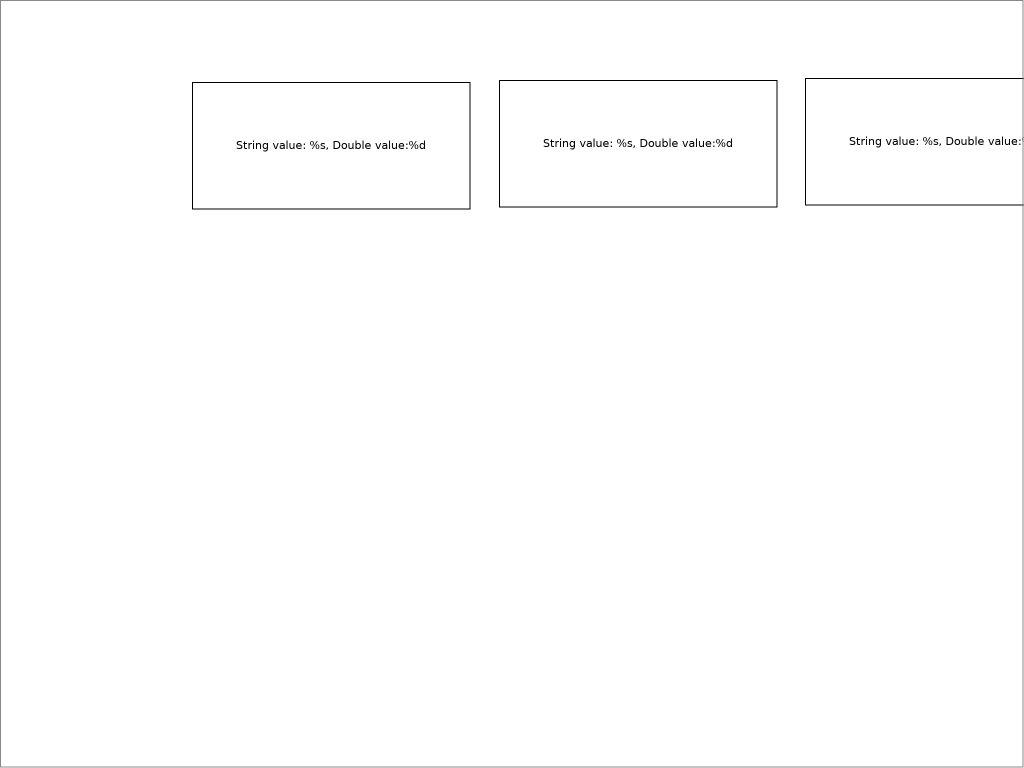
VISUALIZATION Visualization  // 1024x768
    Rectangle (192,82 278x127), "String value: %s, Double value:%d", text variable: MAIN.struct0.sStringProperty
        p4168582468: MAIN.struct0.iNumericProperty
    Rectangle (1110,78 278x127), "String value: %s, Double value:%d", text variable: MAIN.struct3.sStringProperty
        p4168582468: MAIN.struct3.iNumericProperty
    Rectangle (805,78 278x127), "String value: %s, Double value:%d", text variable: MAIN.struct2.sStringProperty
        p4168582468: MAIN.struct2.iNumericProperty
    Rectangle (499,80 278x127), "String value: %s, Double value:%d", text variable: MAIN.struct1.sStringProperty
        p4168582468: MAIN.struct1.iNumericProperty
END_VISUALIZATION

(* stored: Version 1.1.0.1, ProductVersion 3.1.4022.12
   Visu Visualization: Id {68235586-9b56-453a-8da2-909a2384438b} *)
